// TwinCAT 3 PLC project Proje1
// ProgramVersion: 3.1.4024.0
// libraries:
//   Tc2_Standard, * (Beckhoff Automation GmbH)
//   Tc2_System, * (Beckhoff Automation GmbH)
//   Tc2_Utilities, * (Beckhoff Automation GmbH)
//   Tc3_Module, * (Beckhoff Automation GmbH)
// project tree:
//   DUTs/ E_EventType.TcDUT, St_Event.TcDUT
//   / PlcTask.TcTTO
//   POUs/ FB_EventLogger.TcPOU, FB_CsvPersistentEventStorage.TcPOU, I_PersistentEventStorage.TcIO, MAIN.TcPOU, F_UpdateEventTimeStampWithSystemTime.TcPOU

CONFIGURATION Proje1
    RESOURCE PLC ON TwinCAT3
        TASK PlcTask(INTERVAL := T#10ms, PRIORITY := 20);
        PROGRAM MAIN WITH PlcTask : MAIN;
    END_RESOURCE
END_CONFIGURATION

// ---- DUTs/E_EventType.TcDUT
{attribute 'qualified_only'}
{attribute 'strict'}
{attribute 'to_string'}

TYPE E_EventType  :
(
	Alarm := 0,
	Message := 1 
);
END_TYPE

// ---- DUTs/St_Event.TcDUT
TYPE St_Event :
STRUCT
	eEventType : E_EventType ;
	eEventSeverity : TcEventSeverity ;
	nEventIdentiy : UDINT ;
	sEventText : STRING (255) ;
	dtTimeStamp : DATE_AND_TIME ;
	
END_STRUCT
END_TYPE

// ---- POUs/I_PersistentEventStorage.TcIO
INTERFACE I_PersistentEventStorage

METHOD StoreEvent 
VAR_INPUT
	stEvent : St_Event ;
	
END_VAR
END_METHOD

END_INTERFACE

// ---- POUs/MAIN.TcPOU
PROGRAM MAIN
VAR
	//Test : St_Event ;
	buton : BOOL := FALSE ;
	
	eEventType1 : E_EventType := E_EventType.Alarm ;
	eEventSeverity1 : TcEventSeverity := TcEventSeverity.Error ;
	nEventIdentiy1 : UDINT := 42 ;
	sEventText1 : STRING (255) := 'This is a scary event' ;
	
	CsvPersistentEventStorage : FB_CsvPersistentEventStorage ;
	EventLogger : FB_EventLogger(CsvPersistentEventStorage) ;
	
	
END_VAR


IF buton THEN
	EventLogger.AddEvent(eEventType1, eEventSeverity1, nEventIdentiy1, sEventText1);
	buton := FALSE ;
 
END_IF

CsvPersistentEventStorage();

END_PROGRAM

// ---- POUs/FB_CsvPersistentEventStorage.TcPOU
FUNCTION_BLOCK FB_CsvPersistentEventStorage IMPLEMENTS I_PersistentEventStorage
VAR
	fbFileOpen : FB_FileOpen := (sPathName := 'C:\ Events.log' , nMode :=  FOPEN_MODEAPPEND OR FOPEN_MODETEXT ) ;
	fbFilePuts  : FB_FilePuts ;
	fbFileClose : Fb_FileClose ;
	eWriteState : (FILE_OPEN_TRIGGER ,FILE_OPEN , WAIT_FOR_EVENT, WRITE_EVENT_TRIGGER, WRITE_EVENT,FILE_CLOSE_TRIGGER, FILE_CLOSE, ERROR ) ;
	StEventWrittenToFile : St_Event ;
	
	CsvString : T_MaxString ;
	FILE_CLOSE_TRIGGER :INT ;
END_VAR


CASE eWriteState OF
	
	FILE_OPEN_TRIGGER:
		fbFileOpen(bExecute := TRUE ) ;
		eWriteState := FILE_OPEN ;
		
		
	FILE_OPEN 		:
		fbFileOpen(bExecute := FALSE ) ;
		IF fbFileOpen.bError THEN
			eWriteState := ERROR ;
		ELSIF NOT fbFileOpen.bBusy AND fbFileOpen.hFile <> 0 THEN
			eWriteState := WAIT_FOR_EVENT ;	
		END_IF
  	WAIT_FOR_EVENT 	:
	//code yok
	WRITE_EVENT_TRIGGER 	:
		CsvString := CreateCsvString(stEvent := StEventWrittenToFile) ;
		fbFilePuts(bExecute := TRUE,
					sLine := CsvString ,
					hFile := fbFileOpen.hFile) ;
		eWriteState := WRITE_EVENT ;	
		
	WRITE_EVENT 	:
		fbFilePuts(bExecute := FALSE);
		IF fbFilePuts.bError THEN
			eWriteState := ERROR ;
		ELSIF NOT fbFilePuts.bBusy THEN
			eWriteState := WAIT_FOR_EVENT ;
		END_IF
	
	FILE_CLOSE_TRIGGER :
		fbFileClose(bExecute := TRUE ,
				hFile := fbFileOpen.hFile);
		eWriteState := WRITE_EVENT ;
	
	FILE_CLOSE		:
		fbFileClose(bExecute := FALSE ) ;
		IF fbFileClose.bError THEN
			eWriteState := ERROR ;
		ELSIF  NOT fbFileClose.bBusy THEN
			eWriteState := FILE_OPEN_TRIGGER ;
		END_IF
	ERROR :
		//CODE YOK
	
	
END_CASE

METHOD PRIVATE CreateCsvString : T_MaxString
VAR_INPUT
	stEvent : REFERENCE TO ST_EVENt ;
END_VAR
VAR
	TempString : T_MaxString ;
END_VAR
TempString := TO_STRING(stEvent.eEventType) ;
TempString := CONCAT(STR1:= TempString , STR2 := ',') ;
TempString := CONCAT(STR1:= TempString , STR2 := TO_STRING (stEvent.eEventSeverity));
TempString := CONCAT(STR1:= TempString , STR2 := ',') ;
TempString := CONCAT(STR1:= TempString , STR2 := TO_STRING (stEvent.nEventIdentiy )) ;
TempString := CONCAT(STR1:= TempString , STR2 := ',') ;
TempString := CONCAT(STR1:= TempString , STR2 := stEvent.sEventText);
TempString := CONCAT(STR1:= TempString , STR2 := ',') ;
TempString := CONCAT(STR1:= TempString , STR2 := TO_STRING (stEvent.dtTimeStamp)) ;
TempString := CONCAT(STR1:= TempString , STR2 := '$n') ;

CreateCsvString := TempString ;
END_METHOD

{warning 'add method implementation '}
METHOD StoreEvent
VAR_INPUT
	stEvent	: St_Event;
END_VAR
IF eWriteState = WAIT_FOR_EVENT THEN
	eWriteState := Write_EVENT ;
	StEventWrittenToFile := stEvent ;
	
	
END_IF
END_METHOD

END_FUNCTION_BLOCK

// ---- POUs/FB_EventLogger.TcPOU
FUNCTION_BLOCK FB_EventLogger
VAR
 	EventBuffer : ARRAY [1..MAXIMUM_SIZE_OF_EVENT_BUFFER] OF St_Event ;
	CurrentEventBufferIndex : INT := 0 ;
	
	_PersistentEventStorage : I_PersistentEventStorage ;
END_VAR

VAR CONSTANT
	MAXIMUM_SIZE_OF_EVENT_BUFFER : INT := 100 ;
END_VAR



_PersistentEventStorage.StoreEvent(stEvent :=  EventBuffer[CurrentEventBufferIndex]) ;

METHOD PUBLIC AddEvent : BOOL
VAR_INPUT
	eEventType : E_EventType ;
	eEventSeverity : TcEventSeverity ;
	nEventIdentiy : UDINT ;
	sEventText : STRING (255) ;
END_VAR
IF NOT IsEventBufferFull () THEN
	CurrentEventBufferIndex := CurrentEventBufferIndex +1 ;
	EventBuffer[CurrentEventBufferIndex].eEventType 	:= eEventType 		;
	EventBuffer[CurrentEventBufferIndex].eEventSeverity := eEventSeverity 	;
	EventBuffer[CurrentEventBufferIndex].nEventIdentiy 	:= nEventIdentiy	;
	EventBuffer[CurrentEventBufferIndex].sEventText 	:= sEventText		;
	F_UpdateEventTimeStampWithSystemTime(stEvent := EventBuffer[CurrentEventBufferIndex]);
		
	AddEvent := TRUE ;	
ELSE
	AddEvent := FALSE ;
END_IF

_PersistentEventStorage.StoreEvent(stEvent := EventBuffer[CurrentEventBufferIndex]) ;
END_METHOD

METHOD FB_init : BOOL
VAR_INPUT
	bInitRetains : BOOL; // if TRUE, the retain variables are initialized (warm start / cold start)
	bInCopyCode : BOOL;  // if TRUE, the instance afterwards gets moved into the copy code (online change)
	
	iPersistentEventStorage : I_PersistentEventStorage ;
END_VAR

_PersistentEventStorage := iPersistentEventStorage ;
END_METHOD

METHOD PRIVATE IsEventBufferFull : BOOL
VAR_INPUT
	
END_VAR
IF (CurrentEventBufferIndex + 1) > MAXIMUM_SIZE_OF_EVENT_BUFFER THEN
	IsEventBufferFull := TRUE ;
ELSE
	IsEventBufferFull := FALSE ;
END_IF
END_METHOD

END_FUNCTION_BLOCK

// ---- POUs/F_UpdateEventTimeStampWithSystemTime.TcPOU
FUNCTION F_UpdateEventTimeStampWithSystemTime 
VAR_INPUT
	stEvent : REFERENCE TO St_Event ;
END_VAR
VAR
	fbGETSYSTEMTIME : GETSYSTEMTIME ;
	
	stFileTime : T_FILETIME ;
	
END_VAR

fbGETSYSTEMTIME (timeLoDW => stFileTime.dwLowDateTime,
				 timeHiDW => stFileTime.dwHighDateTime) ;
				 
stEvent.dtTimeStamp := FILETIME_TO_DT(fileTime := stFileTime ) ;

END_FUNCTION
